FUNCTION_BLOCK IAS_Skill_StateModel (* Tamplate for a simple Basic Function Block Type *)
  (* Standard: 61499-2 *)
  (* Version 0.0, 2018-05-17, 4DIAC-IDE, 4DIAC-Consortium *)
  (* Version 1.0, 2016-05-26, AZ, fortiss GmbH *)
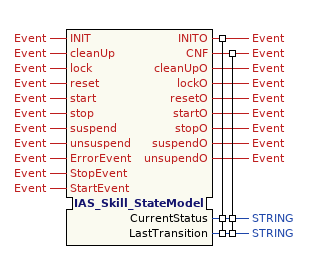
  EVENT_INPUT
    INIT;
    cleanUp; (* Initialization Request *)
    lock; (* Normal Execution Request *)
    reset;
    start;
    stop;
    suspend;
    unsuspend;
    ErrorEvent;
    StopEvent;
    StartEvent;
  END_EVENT
  EVENT_OUTPUT
    INITO WITH CurrentStatus, LastTransition;
    CNF WITH CurrentStatus, LastTransition; (* Execution Confirmation *)
    cleanUpO;
    lockO;
    resetO;
    startO;
    stopO;
    suspendO;
    unsupendO;
  END_EVENT
  VAR_OUTPUT
    CurrentStatus : STRING; (* Output event qualifier *)
    LastTransition : STRING;
  END_VAR
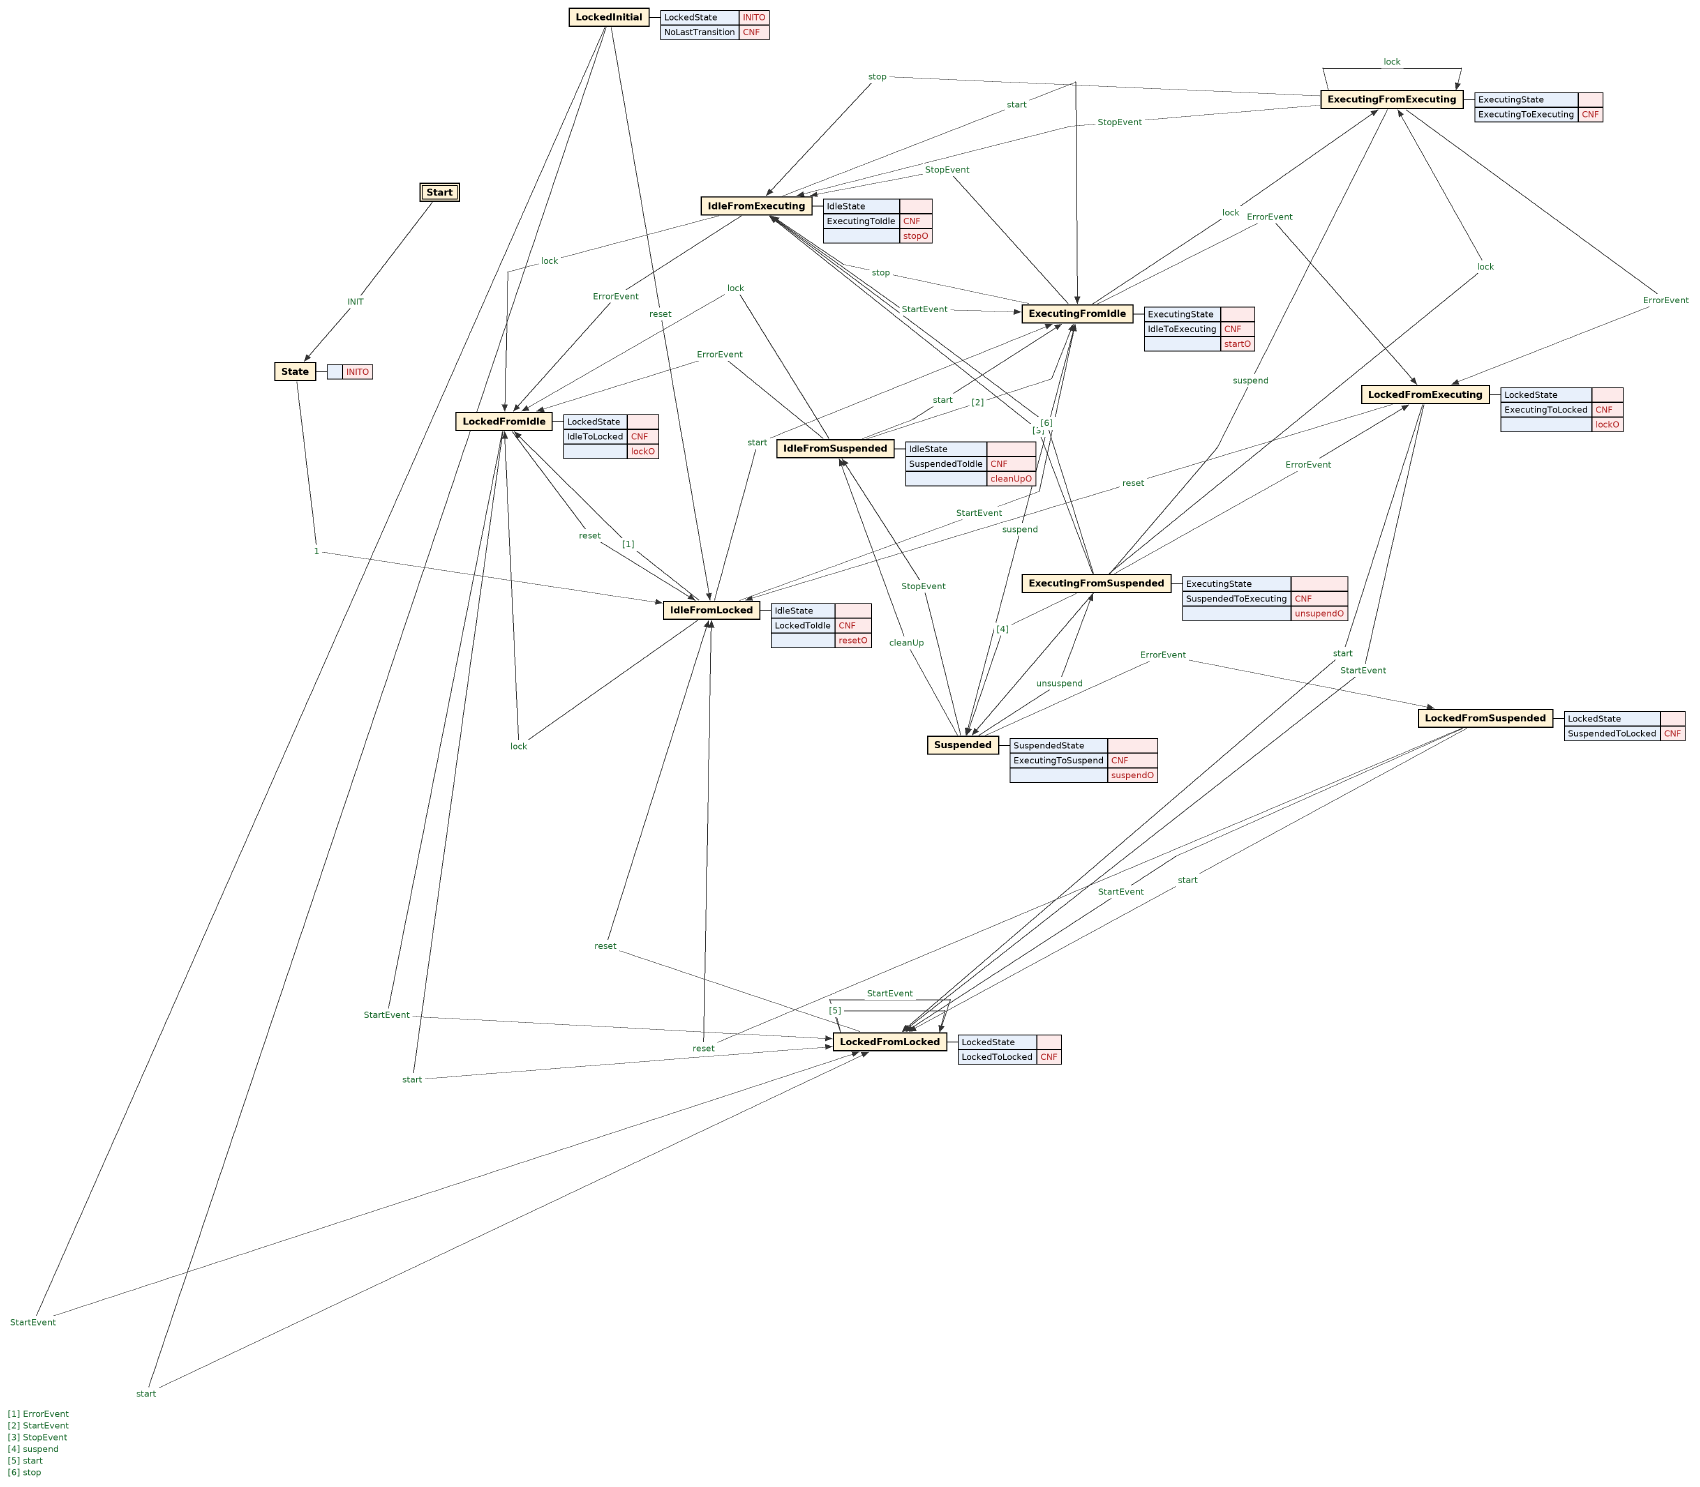
  EC_STATES
    Start; (* Initial State *)
    IdleFromExecuting : IdleState, ExecutingToIdle -> CNF, -> stopO;
    ExecutingFromIdle : ExecutingState, IdleToExecuting -> CNF, -> startO;
    Suspended : SuspendedState, ExecutingToSuspend -> CNF, -> suspendO;
    IdleFromSuspended : IdleState, SuspendedToIdle -> CNF, -> cleanUpO;
    LockedFromExecuting : LockedState, ExecutingToLocked -> CNF, -> lockO;
    LockedFromSuspended : LockedState, SuspendedToLocked -> CNF;
    LockedFromIdle : LockedState, IdleToLocked -> CNF, -> lockO;
    ExecutingFromSuspended : ExecutingState, SuspendedToExecuting -> CNF, -> unsupendO;
    IdleFromLocked : IdleState, LockedToIdle -> CNF, -> resetO;
    LockedInitial : LockedState -> INITO, NoLastTransition -> CNF;
    LockedFromLocked : LockedState, LockedToLocked -> CNF;
    ExecutingFromExecuting : ExecutingState, ExecutingToExecuting -> CNF;
    State : -> INITO;
  END_STATES
  EC_TRANSITIONS
    ExecutingFromIdle TO IdleFromExecuting := stop;
    ExecutingFromSuspended TO IdleFromExecuting := stop;
    ExecutingFromIdle TO LockedFromExecuting := ErrorEvent;
    ExecutingFromSuspended TO LockedFromExecuting := ErrorEvent;
    ExecutingFromSuspended TO Suspended := suspend;
    ExecutingFromIdle TO Suspended := suspend;
    IdleFromExecuting TO ExecutingFromIdle := start;
    IdleFromSuspended TO LockedFromIdle := lock;
    IdleFromExecuting TO LockedFromIdle := lock;
    IdleFromLocked TO ExecutingFromIdle := start;
    IdleFromLocked TO LockedFromIdle := lock;
    LockedFromSuspended TO IdleFromLocked := reset;
    LockedFromExecuting TO IdleFromLocked := reset;
    Suspended TO ExecutingFromSuspended := unsuspend;
    Suspended TO IdleFromSuspended := cleanUp;
    Suspended TO LockedFromSuspended := ErrorEvent;
    IdleFromSuspended TO ExecutingFromIdle := start;
    LockedFromIdle TO LockedFromLocked := start;
    LockedFromSuspended TO LockedFromLocked := start;
    LockedFromExecuting TO LockedFromLocked := start;
    LockedFromLocked TO LockedFromLocked := start;
    LockedFromLocked TO IdleFromLocked := reset;
    ExecutingFromIdle TO ExecutingFromExecuting := lock;
    ExecutingFromSuspended TO ExecutingFromExecuting := lock;
    ExecutingFromExecuting TO IdleFromExecuting := stop;
    ExecutingFromExecuting TO LockedFromExecuting := ErrorEvent;
    ExecutingFromExecuting TO Suspended := suspend;
    ExecutingFromExecuting TO ExecutingFromExecuting := lock;
    LockedInitial TO IdleFromLocked := reset;
    LockedInitial TO LockedFromLocked := start;
    LockedFromIdle TO IdleFromLocked := reset;
    IdleFromSuspended TO LockedFromIdle := ErrorEvent;
    IdleFromExecuting TO LockedFromIdle := ErrorEvent;
    IdleFromLocked TO LockedFromIdle := ErrorEvent;
    Suspended TO IdleFromSuspended := StopEvent;
    ExecutingFromSuspended TO IdleFromExecuting := StopEvent;
    ExecutingFromIdle TO IdleFromExecuting := StopEvent;
    ExecutingFromExecuting TO IdleFromExecuting := StopEvent;
    Start TO State := INIT;
    State TO IdleFromLocked := 1;
    LockedFromLocked TO LockedFromLocked := StartEvent;
    LockedInitial TO LockedFromLocked := StartEvent;
    LockedFromIdle TO LockedFromLocked := StartEvent;
    LockedFromSuspended TO LockedFromLocked := StartEvent;
    LockedFromExecuting TO LockedFromLocked := StartEvent;
    IdleFromLocked TO ExecutingFromIdle := StartEvent;
    IdleFromExecuting TO ExecutingFromIdle := StartEvent;
    IdleFromSuspended TO ExecutingFromIdle := StartEvent;
  END_TRANSITIONS
  ALGORITHM IdleState IN ST: (* Initialization algorithm *)
CurrentStatus := "Idle";
  END_ALGORITHM
  ALGORITHM SuspendedState IN ST: (* Normally executed algorithm *)
CurrentStatus := "Suspended";
  END_ALGORITHM
  ALGORITHM LockedState IN ST: (* new algorithm *)
CurrentStatus := "Locked";
  END_ALGORITHM
  ALGORITHM ExecutingState IN ST: (* new algorithm *)
CurrentStatus := "Executing";
  END_ALGORITHM
  ALGORITHM ExecutingToIdle IN ST: (* new algorithm *)
LastTransition := "ExecutingToIdle";
  END_ALGORITHM
  ALGORITHM ExecutingToLocked IN ST: (* new algorithm *)
LastTransition := "ExecutingToLocked";
  END_ALGORITHM
  ALGORITHM ExecutingToSuspend IN ST: (* new algorithm *)
LastTransition := "ExecutingToSuspend";
  END_ALGORITHM
  ALGORITHM IdleToExecuting IN ST: (* new algorithm *)
LastTransition := "IdleToExecuting";
  END_ALGORITHM
  ALGORITHM IdleToLocked IN ST: (* new algorithm *)
LastTransition := "IdleToLocked";
  END_ALGORITHM
  ALGORITHM LockedToIdle IN ST: (* new algorithm *)
LastTransition := "LockedToIdle";
  END_ALGORITHM
  ALGORITHM SuspendedToExecuting IN ST: (* new algorithm *)
LastTransition := "SuspendedToExecuting";
  END_ALGORITHM
  ALGORITHM SuspendedToIdle IN ST: (* new algorithm *)
LastTransition := "SuspendedToIdle";
  END_ALGORITHM
  ALGORITHM SuspendedToLocked IN ST: (* new algorithm *)
LastTransition := "SuspendedToLocked";
  END_ALGORITHM
  ALGORITHM LockedToLocked IN ST: (* new algorithm *)
LastTransition := "LockedToLocked";
  END_ALGORITHM
  ALGORITHM ExecutingToExecuting IN ST: (* new algorithm *)
LastTransition := "ExecutingToExecuting";
  END_ALGORITHM
  ALGORITHM NoLastTransition IN ST: (* new algorithm *)
LastTransition := "";
  END_ALGORITHM
END_FUNCTION_BLOCK
